INTERFACE I_VolumeFlowController

PROPERTY Error : BOOL
GET
END_GET
SET
END_SET
END_PROPERTY

METHOD Run : BOOL
VAR_INPUT
END_VAR
END_METHOD

PROPERTY VolumeFlowActual : REAL
GET
END_GET
SET
END_SET
END_PROPERTY

PROPERTY VolumeFlowSetpoint : REAL
GET
END_GET
SET
END_SET
END_PROPERTY

END_INTERFACE

(* stored: Version 1.1.0.1, ProductVersion 3.1.4024.0
   Itf I_VolumeFlowController: Id {3e9714a2-8102-406d-bdd7-76b774ef37ff}
   Property Error: Id {0a30ef2f-7548-4dfa-b994-bf245a046028}
   Get Get: Id {e8ea9cf5-e839-4f73-a693-8a38aa5a5390}
   Set Set: Id {737dc09b-3aaf-4bfe-9024-bfcffdf46b35}
   Method Run: Id {9f5bee67-5b89-4245-8540-2f9156157eb3}
   Property VolumeFlowActual: Id {0002fad8-fef2-4c99-b015-31c4d7bab25a}
   Get Get: Id {3aa684af-078b-4c05-8224-28f31fdad097}
   Set Set: Id {a129d950-8d39-4787-b4f3-5f37472a5456}
   Property VolumeFlowSetpoint: Id {62267535-019e-4e05-b11c-3a3b0f2b2f02}
   Get Get: Id {27b70a78-754e-45fe-ab04-e3d133f34bea}
   Set Set: Id {f5befcfd-ec27-4706-a4be-780e2a0657ad} *)
